// SIMATIC S7-200 project (STEP 7-Micro/WIN), CPU 226 CN REL 02.01

SYMBOL_TABLE USER1
Sens_Origen      I0.0     // Sensor inductivo origen servo (usado por libreria MAP_SERV para homing)
FC_Derecha       I0.1     // Final de carrera derecha (Fwd_Limit para Q0_0_CTRL)
FC_Izquierda     I0.2     // Final de carrera izquierda (Rev_Limit para Q0_0_CTRL)
CilV_Abajo       I0.3     // Sensor brazo retraido (abajo)
CilV_Arriba      I0.4     // Sensor brazo extendido (arriba)
Giro_Izquierda   I0.5     // Sensor rotatorio posicion izquierda (antihorario)
Giro_Derecha     I0.6     // Sensor rotatorio posicion derecha (horario)
CilDV_Ext        I0.7     // Sensor doble vastago extendido
CilDV_Ret        I1.0     // Sensor doble vastago retraido
Pinza_Cer        I1.1     // Sensor pinza cerrada
Estado_Servo     I1.2     // Estado driver servo (1=Ready 0=Alarma)
Btn_Paro         I2.4     // Pulsador rojo de paro
Btn_Marcha       I2.5     // Pulsador amarillo de marcha
Seta_Emerg       I2.6     // Seta de emergencia (NC - 0=emergencia activa)
Selector         I2.7     // Selector rotatorio de modo
Servo_Pulsos     Q0.0     // Salida PTO tren de pulsos al driver servo
Servo_Dir        Q0.2     // Salida direccion al driver servo
V_Cil_Vert       Q0.3     // Valvula elevar brazo neumatico (activo=arriba inactivo=baja)
V_Giro_AH        Q0.4     // Valvula rotatorio antihorario (destino Seleccion)
V_Giro_H         Q0.5     // Valvula rotatorio horario (destino Procesamiento y Ensamblaje)
V_Cil_DV         Q0.6     // Valvula doble vastago (extender)
V_Pinza_Abre     Q0.7     // Valvula pinza abre
V_Pinza_Cierra   Q1.0     // Valvula pinza cierra
Lamp_Amarilla    Q1.5     // Lampara amarilla - parada pendiente o homing activo
Lamp_Verde       Q1.6     // Lampara verde - ciclo de tarea en ejecucion
Lamp_Roja        Q1.7     // Lampara roja - reposo esperando solicitud
P_Hom_Espera     M5.0     // Plaza Homing_Espera - estado inicial al arranque o tras emergencia
P_Hom_Activo     M5.1     // Plaza Homing_Activo - servo buscando origen
P0_Brazo_Libre   M0.0     // Plaza P0 - Reposo. Brazo disponible para nueva tarea
P1_Req_A_P       M0.1     // Plaza P1 - Solicitud activa Alimentacion -> Procesamiento (inyectable Modbus)
P2_Req_P_E       M0.2     // Plaza P2 - Solicitud activa Procesamiento -> Ensamblaje (inyectable Modbus)
P3_Req_E_S       M0.3     // Plaza P3 - Solicitud activa Ensamblaje -> Seleccion (inyectable Modbus)
P10_Viaje_Ori    M1.0     // Plaza P10 - Servo viajando a coordenada de recogida
P11a_Rot_Ori     M1.1     // Plaza P11a - Orientando garra en posicion de recogida
P11b_DV_Ext      M1.2     // Plaza P11b - Extendiendo doble vastago en pick
P11c_Cil_Baj     M1.3     // Plaza P11c - Bajando brazo en pick
P11d_Pinza_Cer   M1.4     // Plaza P11d - Cerrando pinza (agarrando pieza)
P11e_Cil_Arr     M1.5     // Plaza P11e - Subiendo brazo con pieza
P11f_DV_Ret      M1.6     // Plaza P11f - Retrayendo doble vastago (pick completo)
P12_Viaje_Des    M1.7     // Plaza P12 - Servo viajando a coordenada de entrega
P13a_Rot_Des     M2.0     // Plaza P13a - Orientando garra en posicion de entrega
P13b_DV_Ext      M2.1     // Plaza P13b - Extendiendo doble vastago en place
P13c_Cil_Baj     M2.2     // Plaza P13c - Bajando brazo en place
P13d_Pinza_Ab    M8.0     // Plaza P13d - Abriendo pinza (liberando pieza)
P13e_Cil_Arr     M8.1     // Plaza P13e - Subiendo brazo tras soltar
P13f_DV_Ret      M3.5     // Plaza P13f - Retrayendo doble vastago (place completo)
P14_Finalizar    M3.6     // Plaza P14 - Liberando brazo y limpiando solicitud
Ev_Marcha_Flanco M6.0     // Evento - Flanco subida boton marcha (autorreset en P0)
Ev_Paro_Flanco   M6.1     // Evento - Flanco subida boton paro (bloquea inicio nuevo ciclo)
Ev_CilV_Abajo    M2.3     // Evento - Sensor brazo abajo
Ev_CilV_Arriba   M2.4     // Evento - Sensor brazo arriba
Ev_Giro_Izq      M2.5     // Evento - Sensor rotatorio posicion izquierda
Ev_Giro_Der      M2.6     // Evento - Sensor rotatorio posicion derecha (horario)
Ev_CilDV_Ext     M2.7     // Evento - Sensor doble vastago extendido
Ev_CilDV_Ret     M3.0     // Evento - Sensor doble vastago retraido
Ev_Pinza_Cer     M3.1     // Evento - Pinza cerrada
Ev_Move_Done     M3.2     // Evento - Flag Done libreria MAP_SERV (posicion alcanzada)
Ev_Origen_Det    M3.3     // Evento - Sensor I0.0 origen detectado (usado en homing)
Ev_Servo_OK      M3.4     // Evento - Driver servo listo (I1.2=1)
T_Homing_Start   M4.0     // Disparo - Iniciar secuencia de homing
T_Homing_Done    M4.1     // Disparo - Homing completado sensor origen detectado
T_Acept_ES       M4.2     // Disparo - Aceptar tarea E->S (Prioridad 1 alta)
T_Acept_PE       M4.3     // Disparo - Aceptar tarea P->E (Prioridad 2 media)
T_Acept_AP       M4.4     // Disparo - Aceptar tarea A->P (Prioridad 3 baja)
T_Origen_OK      M4.5     // Disparo - Servo llego a coordenada de recogida
T_Rot_Ori_OK     M4.6     // Disparo - Garra orientada en posicion de recogida
T_DV_Ext_Pick    M4.7     // Disparo - Doble vastago extendido en pick
T_CilV_Baj_Pick  M5.2     // Disparo - Brazo abajo en pick
T_Pinza_Cer      M5.3     // Disparo - Pinza cerrada agarre confirmado
T_CilV_Arr_Pick  M5.4     // Disparo - Brazo arriba con pieza en pick
T_DV_Ret_Pick    M5.5     // Disparo - Doble vastago retraido pick completo
T_Destino_OK     M5.6     // Disparo - Servo llego a coordenada de entrega
T_Rot_Des_OK     M5.7     // Disparo - Garra orientada en posicion de entrega
T_DV_Ext_Place   M6.2     // Disparo - Doble vastago extendido en place
T_CilV_Baj_Place M6.3     // Disparo - Brazo abajo en place
T_Pinza_Ab       M6.4     // Disparo - Pinza abierta pieza liberada
T_CilV_Arr_Place M6.5     // Disparo - Brazo arriba tras soltar en place
T_DV_Ret_Place   M6.6     // Disparo - Doble vastago retraido place completo
T_Tarea_Fin      M6.7     // Disparo - Liberar brazo y volver a reposo
Ctx_Tarea_AP     M7.0     // Contexto tarea activa - Alimentacion -> Procesamiento
Ctx_Tarea_PE     M7.1     // Contexto tarea activa - Procesamiento -> Ensamblaje
Ctx_Tarea_ES     M7.2     // Contexto tarea activa - Ensamblaje -> Seleccion
Home_Done        V221.0   // Bit Done libreria MAP_SERV (busqueda de origen alcanzada)
Home_error       V221.1   // Bit Error libreria MAP_SERV (avisa si hubo un error en la busqueda de origen)
Servo_Exec       V220.0   // Bit interno - Comando ejecutar movimiento (nivel)
Servo_Done       V220.1   // Bit Done libreria MAP_SERV (posicion alcanzada)
Servo_Err        V220.2   // Bit Error libreria MAP_SERV
Servo_Execute_Pulse V220.4   // Bit pulso EXECUTE un scan para MoveAbsolute
Servo_C_Pos      VD34     // Posicion actual del servo en pulsos (salida Q0_0_CTRL)
Coord_Target     VD200    // Coordenada destino activa cargada antes de MoveAbsolute
Coord_Alim       VD204    // Coordenada estacion Alimentacion (pulsos)
Coord_Proc       VD208    // Coordenada estacion Procesamiento (pulsos)
Coord_Ensa       VD212    // Coordenada estacion Ensamblaje (pulsos)
Coord_Sele       VD216    // Coordenada estacion Seleccion (pulsos)
net_cycle        M10.0    // network cycle (PPI)
net_error        M10.1    // network error (PPI)
done_modbus      M10.2    // marca done para libreria modbus (init)
error_modbus     VB26     // byte de error para libreria modbus (init)
done_modbus2     M10.3    // marca done para libreria modbus
error_modbus2    VB30     // byte de error para libreria modbus
Pos_Alim         VD10     // Posicion Alimentacion (buffer para la carga dinamica de la posicion)
Pos_Proc         VD14     // Posicion Procesamiento (buffer para la carga dinamica de la posicion)
Pos_Ensa         VD18     // Posicion Ensamblaje (buffer para la carga dinamica de la posicion)
Pos_Sele         VD22     // Posicion Seleccion (buffer para la carga dinamica de la posicion)
Sol_AP           V0.0     // Solicitud Alimentacion a Procesamiento
Ack_AP           V1.0     // Reconocimiento AP
Sol_PE           V2.0     // Solicitud Procesamiento a Ensamblaje
Ack_PE           V3.0     // Reconocimiento PE
Sol_ES           V4.0     // Solicitud Ensamblaje a Seleccion
Ack_ES           V5.0     // Reconocimiento ES
Ack_MA           V0.1     // Reconocimiento marcha Unidad de Alimentacion
Marcha_A         V1.1     // Solicitud de marcha para la Unidad de Alimentacion
Ack_MP           V2.1     // Reconocimiento marcha Unidad de Procesammiento
Marcha_P         V3.1     // Solicitud de marcha para la Unidad de Procesamiento
Ack_ME           V4.1     // Reconocimiento marcha Unidad de Ensamblaje
Marcha_E         V5.1     // Solicitud de marcha para la Unidad de Ensamblaje
Ack_MS           V6.1     // Reconocimiento marcha Unidad de Seleccion
Marcha_S         V7.1     // Solicitud de marcha para la Unidad de Seleccion
Alim_OK          V0.2     // Unidad de Alimentacion disponible
Proc_OK          V2.2     // Unidad de Procesamiento disponible
Ens_OK           V4.2     // Unidad de Ensamblaje disponible
Sel_OK           V6.2     // Unidad de Seleccion disponible
Pieza_Metal      V6.3     // Pieza identificada por la unidad de seleccion es totalmente metalica
Pieza_Mixta      V6.4     // Pieza identificada por la unidad de seleccion es totalmente mixta
Pieza_Plastica   V6.5     // Pieza identificada por la unidad de seleccion es totalmente plastica
END_SYMBOL_TABLE

SYMBOL_TABLE S7-200 Symbols
Always_On        SM0.0    // 始终接通为 ON
First_Scan_On    SM0.1    // 仅第一个扫描周期中接通为 ON
END_SYMBOL_TABLE

ORGANIZATION_BLOCK MAIN:OB1
TITLE=UNIDAD DE TRANSPORTE - RED DE PETRI CIPN
//  ===========================================================
//  MODULO 0: SEGURIDAD - Evaluado primero en cada scan.
//  Si Seta = 0 (NC abierta): reset total, fuerza P_Homing,
//  apaga salidas neumaticas. El servo se detiene porque
//  Q0_0_CTRL deja de recibir EXECUTE.
//  ===========================================================
BEGIN
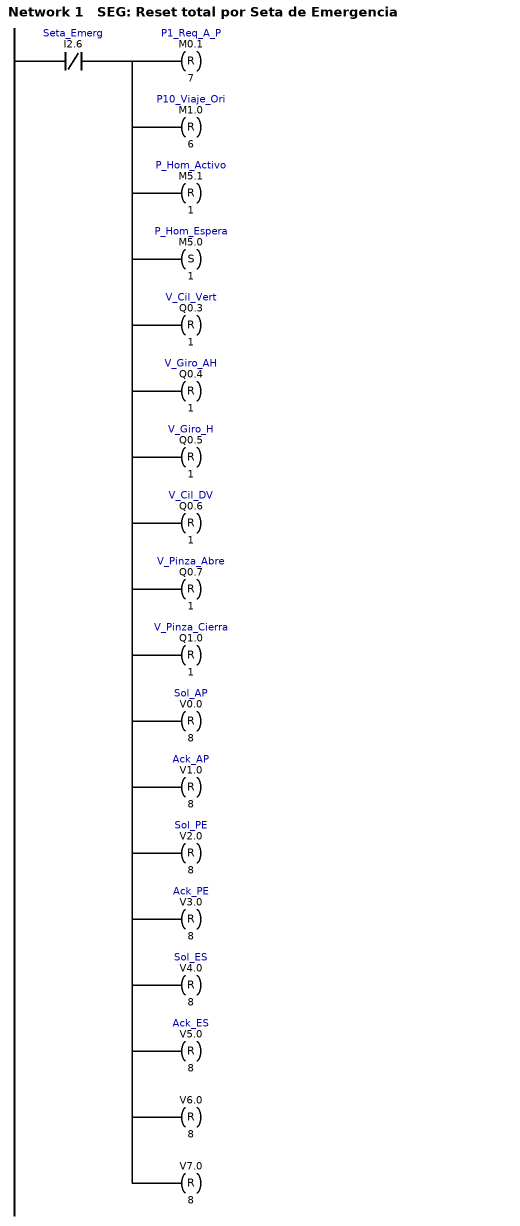
Network 1 //  SEG: Reset total por Seta de Emergencia
LDN    Seta_Emerg:I2.6
R      P1_Req_A_P:M0.1, 7
R      P10_Viaje_Ori:M1.0, 6
R      P_Hom_Activo:M5.1, 1
S      P_Hom_Espera:M5.0, 1
R      V_Cil_Vert:Q0.3, 1
R      V_Giro_AH:Q0.4, 1
R      V_Giro_H:Q0.5, 1
R      V_Cil_DV:Q0.6, 1
R      V_Pinza_Abre:Q0.7, 1
R      V_Pinza_Cierra:Q1.0, 1
R      Sol_AP:V0.0, 8
R      Ack_AP:V1.0, 8
R      Sol_PE:V2.0, 8
R      Ack_PE:V3.0, 8
R      Sol_ES:V4.0, 8
R      Ack_ES:V5.0, 8
R      V6.0, 8
R      V7.0, 8
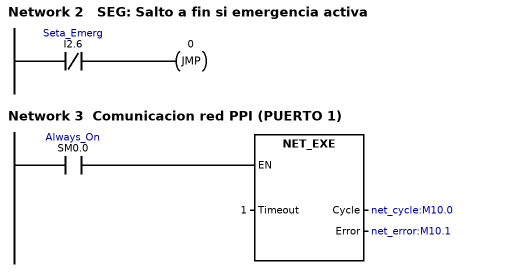
Network 2 //  SEG: Salto a fin si emergencia activa
LDN    Seta_Emerg:I2.6
JMP    0
Network 3 // Comunicacion red PPI (PUERTO 1)
LD     Always_On:SM0.0
CALL   NET_EXE:SBR6, 1, net_cycle:M10.0, net_error:M10.1
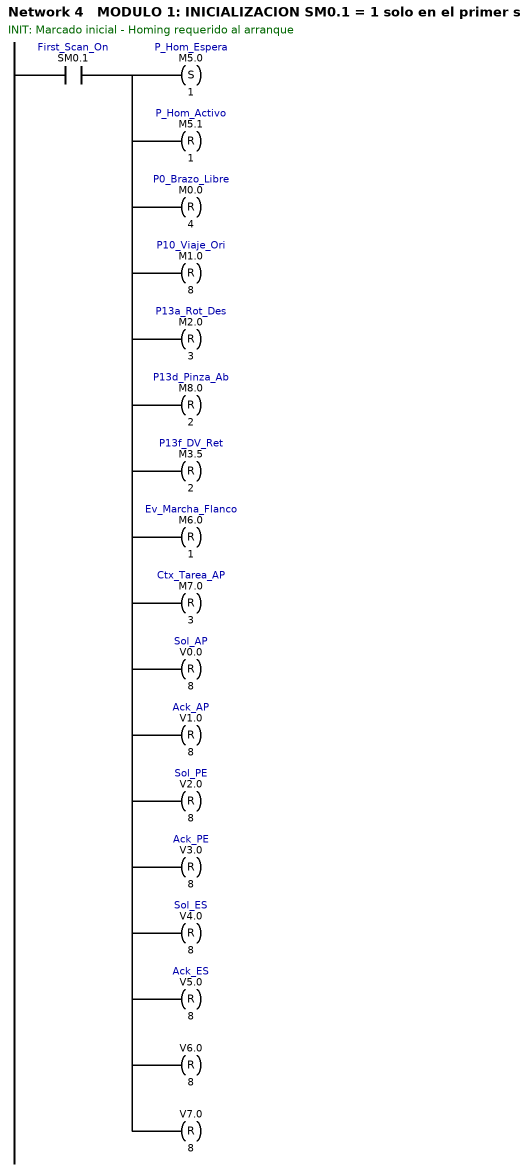
Network 4 //  MODULO 1: INICIALIZACION
SM0.1 = 1 solo en el primer scan.
Marcado inicial: P_Homing activo (M5.0).
El brazo debe calibrarse antes de aceptar cualquier tarea.
Coordenadas de estaciones cargadas en VD fijos.
// INIT: Marcado inicial - Homing requerido al arranque
LD     First_Scan_On:SM0.1
S      P_Hom_Espera:M5.0, 1
R      P_Hom_Activo:M5.1, 1
R      P0_Brazo_Libre:M0.0, 4
R      P10_Viaje_Ori:M1.0, 8
R      P13a_Rot_Des:M2.0, 3
R      P13d_Pinza_Ab:M8.0, 2
R      P13f_DV_Ret:M3.5, 2
R      Ev_Marcha_Flanco:M6.0, 1
R      Ctx_Tarea_AP:M7.0, 3
R      Sol_AP:V0.0, 8
R      Ack_AP:V1.0, 8
R      Sol_PE:V2.0, 8
R      Ack_PE:V3.0, 8
R      Sol_ES:V4.0, 8
R      Ack_ES:V5.0, 8
R      V6.0, 8
R      V7.0, 8
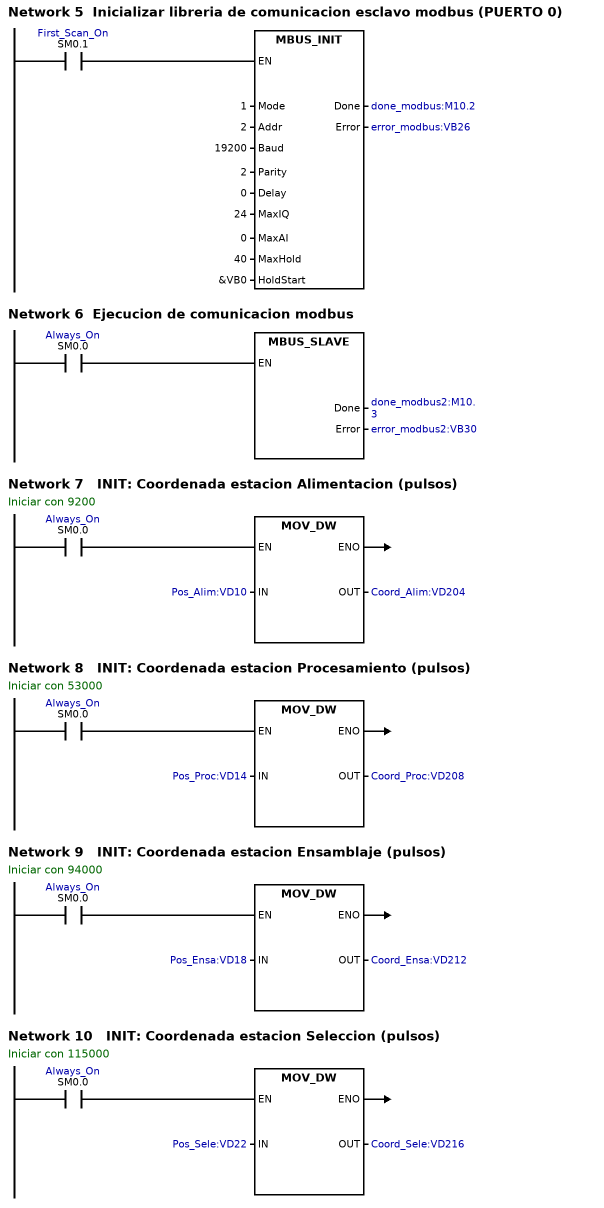
Network 5 // Inicializar libreria de comunicacion esclavo modbus (PUERTO 0)
LD     First_Scan_On:SM0.1
CALL   MBUS_INIT:SBR7, 1, 2, 19200, 2, 0, 24, 0, 40, &VB0, done_modbus:M10.2, error_modbus:VB26
Network 6 // Ejecucion de comunicacion modbus
LD     Always_On:SM0.0
CALL   MBUS_SLAVE:SBR8, done_modbus2:M10.3, error_modbus2:VB30
Network 7 //  INIT: Coordenada estacion Alimentacion (pulsos)
// Iniciar con 9200
LD     Always_On:SM0.0
MOVD   Pos_Alim:VD10, Coord_Alim:VD204
Network 8 //  INIT: Coordenada estacion Procesamiento (pulsos)
// Iniciar con 53000
LD     Always_On:SM0.0
MOVD   Pos_Proc:VD14, Coord_Proc:VD208
Network 9 //  INIT: Coordenada estacion Ensamblaje (pulsos)
// Iniciar con 94000
LD     Always_On:SM0.0
MOVD   Pos_Ensa:VD18, Coord_Ensa:VD212
Network 10 //  INIT: Coordenada estacion Seleccion (pulsos)
// Iniciar con 115000
LD     Always_On:SM0.0
MOVD   Pos_Sele:VD22, Coord_Sele:VD216
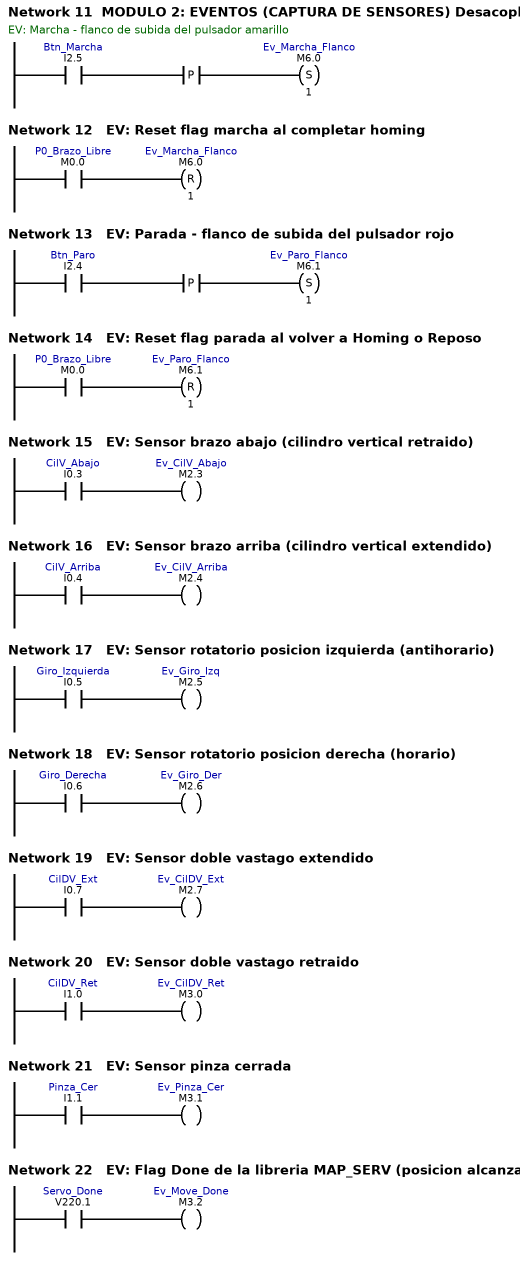
Network 11 // MODULO 2: EVENTOS (CAPTURA DE SENSORES)
Desacopla la logica secuencial de las senales fisicas.
M5.x reservado para estados de Homing y sistema.
M2.x / M3.x para eventos de sensores.
// EV: Marcha - flanco de subida del pulsador amarillo
LD     Btn_Marcha:I2.5
EU
S      Ev_Marcha_Flanco:M6.0, 1
Network 12 //  EV: Reset flag marcha al completar homing
LD     P0_Brazo_Libre:M0.0
R      Ev_Marcha_Flanco:M6.0, 1
Network 13 //  EV: Parada - flanco de subida del pulsador rojo
LD     Btn_Paro:I2.4
EU
S      Ev_Paro_Flanco:M6.1, 1
Network 14 //  EV: Reset flag parada al volver a Homing o Reposo
LD     P0_Brazo_Libre:M0.0
R      Ev_Paro_Flanco:M6.1, 1
Network 15 //  EV: Sensor brazo abajo (cilindro vertical retraido)
LD     CilV_Abajo:I0.3
=      Ev_CilV_Abajo:M2.3
Network 16 //  EV: Sensor brazo arriba (cilindro vertical extendido)
LD     CilV_Arriba:I0.4
=      Ev_CilV_Arriba:M2.4
Network 17 //  EV: Sensor rotatorio posicion izquierda (antihorario)
LD     Giro_Izquierda:I0.5
=      Ev_Giro_Izq:M2.5
Network 18 //  EV: Sensor rotatorio posicion derecha (horario)
LD     Giro_Derecha:I0.6
=      Ev_Giro_Der:M2.6
Network 19 //  EV: Sensor doble vastago extendido
LD     CilDV_Ext:I0.7
=      Ev_CilDV_Ext:M2.7
Network 20 //  EV: Sensor doble vastago retraido
LD     CilDV_Ret:I1.0
=      Ev_CilDV_Ret:M3.0
Network 21 //  EV: Sensor pinza cerrada
LD     Pinza_Cer:I1.1
=      Ev_Pinza_Cer:M3.1
Network 22 //  EV: Flag Done de la libreria MAP_SERV (posicion alcanzada)
LD     Servo_Done:V220.1
=      Ev_Move_Done:M3.2
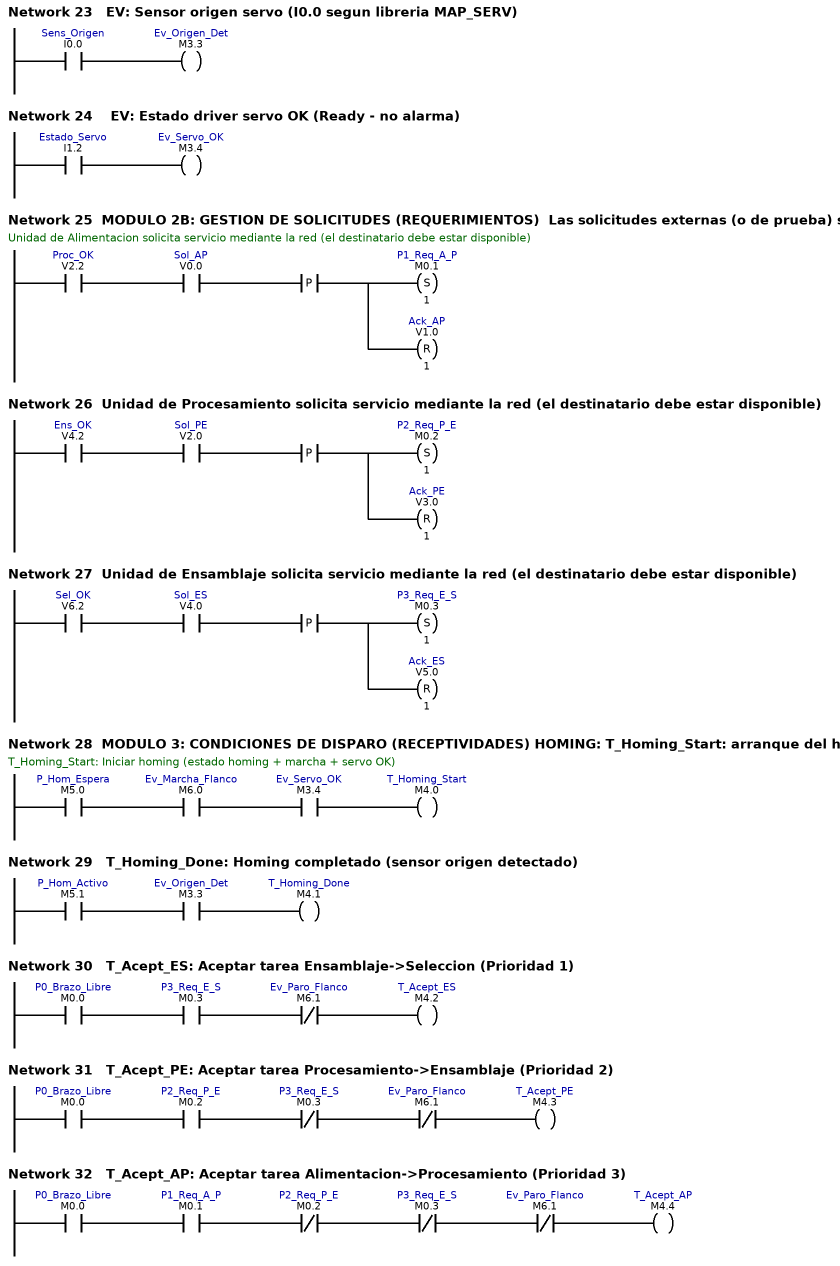
Network 23 //  EV: Sensor origen servo (I0.0 segun libreria MAP_SERV)
LD     Sens_Origen:I0.0
=      Ev_Origen_Det:M3.3
Network 24 //   EV: Estado driver servo OK (Ready - no alarma)
LD     Estado_Servo:I1.2
=      Ev_Servo_OK:M3.4
Network 25 // MODULO 2B: GESTION DE SOLICITUDES (REQUERIMIENTOS)
 Las solicitudes externas (o de prueba) se inyectan en
 M0.1, M0.2, M0.3 desde fuera (Modbus, HMI, o prueba manual).
 Este bloque las protege: solo se aceptan si el sistema
 esta en Reposo (P0 = M0.0 activo)
// Unidad de Alimentacion solicita servicio mediante la red (el destinatario debe estar disponible)
LD     Proc_OK:V2.2
A      Sol_AP:V0.0
EU
S      P1_Req_A_P:M0.1, 1
R      Ack_AP:V1.0, 1
Network 26 // Unidad de Procesamiento solicita servicio mediante la red (el destinatario debe estar disponible)
LD     Ens_OK:V4.2
A      Sol_PE:V2.0
EU
S      P2_Req_P_E:M0.2, 1
R      Ack_PE:V3.0, 1
Network 27 // Unidad de Ensamblaje solicita servicio mediante la red (el destinatario debe estar disponible)
LD     Sel_OK:V6.2
A      Sol_ES:V4.0
EU
S      P3_Req_E_S:M0.3, 1
R      Ack_ES:V5.0, 1
Network 28 // MODULO 3: CONDICIONES DE DISPARO (RECEPTIVIDADES)
HOMING:
T_Homing_Start: arranque del homing (marcha presionada)
T_Homing_Done:  sensor origen detectado
ACEPTACION DE TAREA (priorizadas, mutuamente excluyentes):
T_Acept_ES: P0 AND P3           (Prioridad 1 - Alta)
T_Acept_PE: P0 AND P2 AND !P3   (Prioridad 2 - Media)
T_Acept_AP: P0 AND P1 AND !P2 !P3 (Prioridad 3 - Baja)
CICLO DE TAREA:
Sub-plazas Pick (P11a..P11e) y Place (P13a..P13e)
para modelar los 5 pasos de cada secuencia.
//  T_Homing_Start: Iniciar homing (estado homing + marcha + servo OK)
LD     P_Hom_Espera:M5.0
A      Ev_Marcha_Flanco:M6.0
A      Ev_Servo_OK:M3.4
=      T_Homing_Start:M4.0
Network 29 //  T_Homing_Done: Homing completado (sensor origen detectado)
LD     P_Hom_Activo:M5.1
A      Ev_Origen_Det:M3.3
=      T_Homing_Done:M4.1
Network 30 //  T_Acept_ES: Aceptar tarea Ensamblaje->Seleccion (Prioridad 1)
LD     P0_Brazo_Libre:M0.0
A      P3_Req_E_S:M0.3
AN     Ev_Paro_Flanco:M6.1
=      T_Acept_ES:M4.2
Network 31 //  T_Acept_PE: Aceptar tarea Procesamiento->Ensamblaje (Prioridad 2)
LD     P0_Brazo_Libre:M0.0
A      P2_Req_P_E:M0.2
AN     P3_Req_E_S:M0.3
AN     Ev_Paro_Flanco:M6.1
=      T_Acept_PE:M4.3
Network 32 //  T_Acept_AP: Aceptar tarea Alimentacion->Procesamiento (Prioridad 3)
LD     P0_Brazo_Libre:M0.0
A      P1_Req_A_P:M0.1
AN     P2_Req_P_E:M0.2
AN     P3_Req_E_S:M0.3
AN     Ev_Paro_Flanco:M6.1
=      T_Acept_AP:M4.4
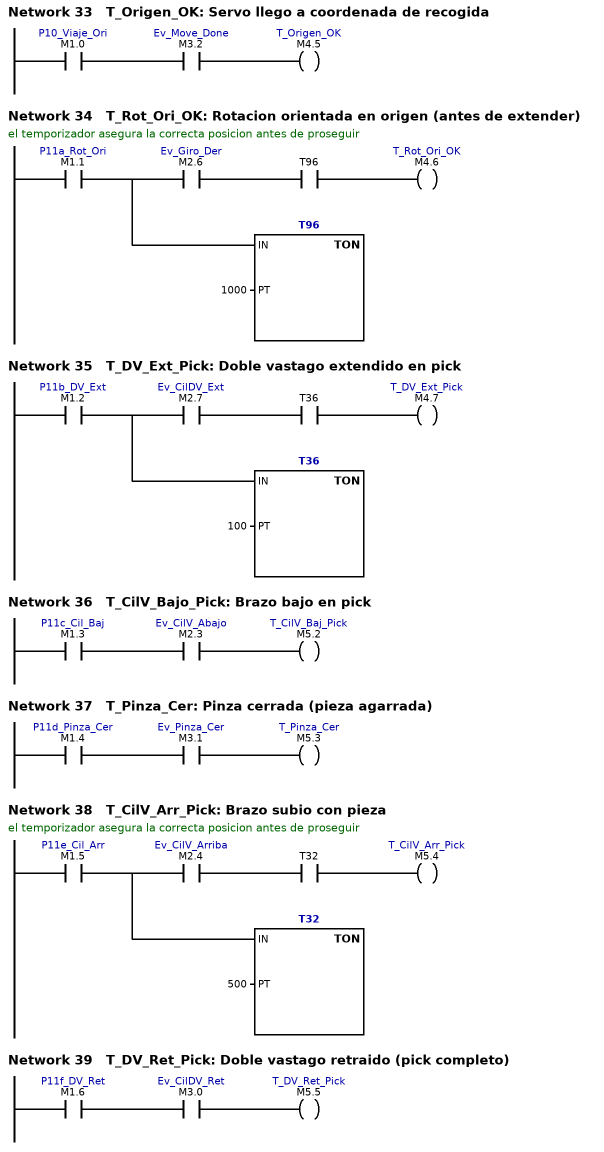
Network 33 //  T_Origen_OK: Servo llego a coordenada de recogida
LD     P10_Viaje_Ori:M1.0
A      Ev_Move_Done:M3.2
=      T_Origen_OK:M4.5
Network 34 //  T_Rot_Ori_OK: Rotacion orientada en origen (antes de extender)
// el temporizador asegura la correcta posicion antes de proseguir
LD     P11a_Rot_Ori:M1.1
LPS
A      Ev_Giro_Der:M2.6
A      T96
=      T_Rot_Ori_OK:M4.6
LPP
TON    T96, 1000
Network 35 //  T_DV_Ext_Pick: Doble vastago extendido en pick
LD     P11b_DV_Ext:M1.2
LPS
A      Ev_CilDV_Ext:M2.7
A      T36
=      T_DV_Ext_Pick:M4.7
LPP
TON    T36, 100
Network 36 //  T_CilV_Bajo_Pick: Brazo bajo en pick
LD     P11c_Cil_Baj:M1.3
A      Ev_CilV_Abajo:M2.3
=      T_CilV_Baj_Pick:M5.2
Network 37 //  T_Pinza_Cer: Pinza cerrada (pieza agarrada)
LD     P11d_Pinza_Cer:M1.4
A      Ev_Pinza_Cer:M3.1
=      T_Pinza_Cer:M5.3
Network 38 //  T_CilV_Arr_Pick: Brazo subio con pieza
// el temporizador asegura la correcta posicion antes de proseguir
LD     P11e_Cil_Arr:M1.5
LPS
A      Ev_CilV_Arriba:M2.4
A      T32
=      T_CilV_Arr_Pick:M5.4
LPP
TON    T32, 500
Network 39 //  T_DV_Ret_Pick: Doble vastago retraido (pick completo)
LD     P11f_DV_Ret:M1.6
A      Ev_CilDV_Ret:M3.0
=      T_DV_Ret_Pick:M5.5
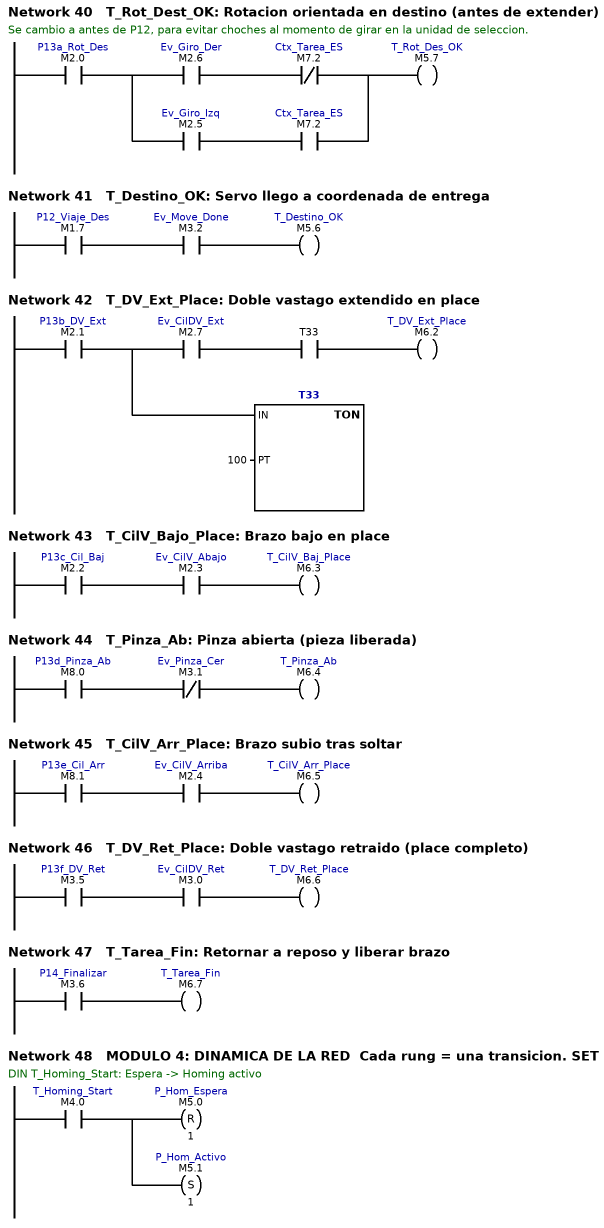
Network 40 //  T_Rot_Dest_OK: Rotacion orientada en destino (antes de extender)
// Se cambio a antes de P12, para evitar choches al momento de girar en la unidad de seleccion.
LD     P13a_Rot_Des:M2.0
LD     Ev_Giro_Der:M2.6
AN     Ctx_Tarea_ES:M7.2
LD     Ev_Giro_Izq:M2.5
A      Ctx_Tarea_ES:M7.2
OLD
ALD
=      T_Rot_Des_OK:M5.7
Network 41 //  T_Destino_OK: Servo llego a coordenada de entrega
LD     P12_Viaje_Des:M1.7
A      Ev_Move_Done:M3.2
=      T_Destino_OK:M5.6
Network 42 //  T_DV_Ext_Place: Doble vastago extendido en place
LD     P13b_DV_Ext:M2.1
LPS
A      Ev_CilDV_Ext:M2.7
A      T33
=      T_DV_Ext_Place:M6.2
LPP
TON    T33, 100
Network 43 //  T_CilV_Bajo_Place: Brazo bajo en place
LD     P13c_Cil_Baj:M2.2
A      Ev_CilV_Abajo:M2.3
=      T_CilV_Baj_Place:M6.3
Network 44 //  T_Pinza_Ab: Pinza abierta (pieza liberada)
LD     P13d_Pinza_Ab:M8.0
AN     Ev_Pinza_Cer:M3.1
=      T_Pinza_Ab:M6.4
Network 45 //  T_CilV_Arr_Place: Brazo subio tras soltar
LD     P13e_Cil_Arr:M8.1
A      Ev_CilV_Arriba:M2.4
=      T_CilV_Arr_Place:M6.5
Network 46 //  T_DV_Ret_Place: Doble vastago retraido (place completo)
LD     P13f_DV_Ret:M3.5
A      Ev_CilDV_Ret:M3.0
=      T_DV_Ret_Place:M6.6
Network 47 //  T_Tarea_Fin: Retornar a reposo y liberar brazo
//  
LD     P14_Finalizar:M3.6
=      T_Tarea_Fin:M6.7
Network 48 //  MODULO 4: DINAMICA DE LA RED
 Cada rung = una transicion. SET destino, RESET origen.
 El marcado de contexto (cual solicitud se esta atendiendo)
 se guarda en M7.0 (es A->P), M7.1 (es P->E), M7.2 (es E->S).
 La orientacion de garra se decide por M7.2 (Seleccion=AH).
// DIN T_Homing_Start: Espera -> Homing activo
LD     T_Homing_Start:M4.0
R      P_Hom_Espera:M5.0, 1
S      P_Hom_Activo:M5.1, 1
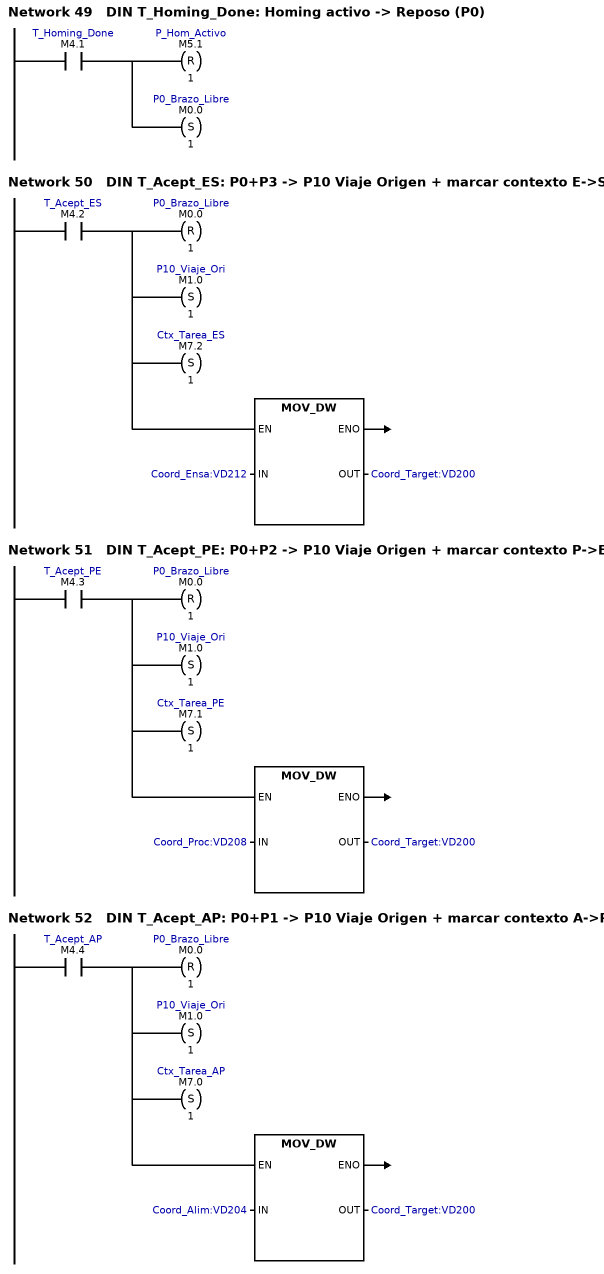
Network 49 //  DIN T_Homing_Done: Homing activo -> Reposo (P0)
LD     T_Homing_Done:M4.1
R      P_Hom_Activo:M5.1, 1
S      P0_Brazo_Libre:M0.0, 1
Network 50 //  DIN T_Acept_ES: P0+P3 -> P10 Viaje Origen + marcar contexto E->S
LD     T_Acept_ES:M4.2
R      P0_Brazo_Libre:M0.0, 1
S      P10_Viaje_Ori:M1.0, 1
S      Ctx_Tarea_ES:M7.2, 1
MOVD   Coord_Ensa:VD212, Coord_Target:VD200
Network 51 //  DIN T_Acept_PE: P0+P2 -> P10 Viaje Origen + marcar contexto P->E
LD     T_Acept_PE:M4.3
R      P0_Brazo_Libre:M0.0, 1
S      P10_Viaje_Ori:M1.0, 1
S      Ctx_Tarea_PE:M7.1, 1
MOVD   Coord_Proc:VD208, Coord_Target:VD200
Network 52 //  DIN T_Acept_AP: P0+P1 -> P10 Viaje Origen + marcar contexto A->P
LD     T_Acept_AP:M4.4
R      P0_Brazo_Libre:M0.0, 1
S      P10_Viaje_Ori:M1.0, 1
S      Ctx_Tarea_AP:M7.0, 1
MOVD   Coord_Alim:VD204, Coord_Target:VD200
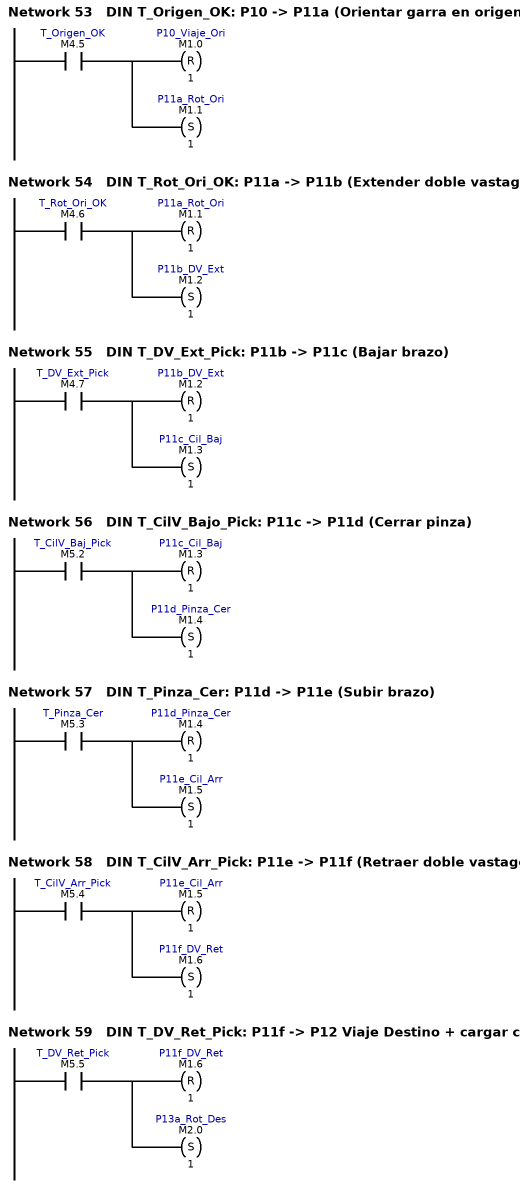
Network 53 //  DIN T_Origen_OK: P10 -> P11a (Orientar garra en origen)
LD     T_Origen_OK:M4.5
R      P10_Viaje_Ori:M1.0, 1
S      P11a_Rot_Ori:M1.1, 1
Network 54 //  DIN T_Rot_Ori_OK: P11a -> P11b (Extender doble vastago)
LD     T_Rot_Ori_OK:M4.6
R      P11a_Rot_Ori:M1.1, 1
S      P11b_DV_Ext:M1.2, 1
Network 55 //  DIN T_DV_Ext_Pick: P11b -> P11c (Bajar brazo)
LD     T_DV_Ext_Pick:M4.7
R      P11b_DV_Ext:M1.2, 1
S      P11c_Cil_Baj:M1.3, 1
Network 56 //  DIN T_CilV_Bajo_Pick: P11c -> P11d (Cerrar pinza)
LD     T_CilV_Baj_Pick:M5.2
R      P11c_Cil_Baj:M1.3, 1
S      P11d_Pinza_Cer:M1.4, 1
Network 57 //  DIN T_Pinza_Cer: P11d -> P11e (Subir brazo)
LD     T_Pinza_Cer:M5.3
R      P11d_Pinza_Cer:M1.4, 1
S      P11e_Cil_Arr:M1.5, 1
Network 58 //  DIN T_CilV_Arr_Pick: P11e -> P11f (Retraer doble vastago)
LD     T_CilV_Arr_Pick:M5.4
R      P11e_Cil_Arr:M1.5, 1
S      P11f_DV_Ret:M1.6, 1
Network 59 //  DIN T_DV_Ret_Pick: P11f -> P12 Viaje Destino + cargar coord destino
LD     T_DV_Ret_Pick:M5.5
R      P11f_DV_Ret:M1.6, 1
S      P13a_Rot_Des:M2.0, 1
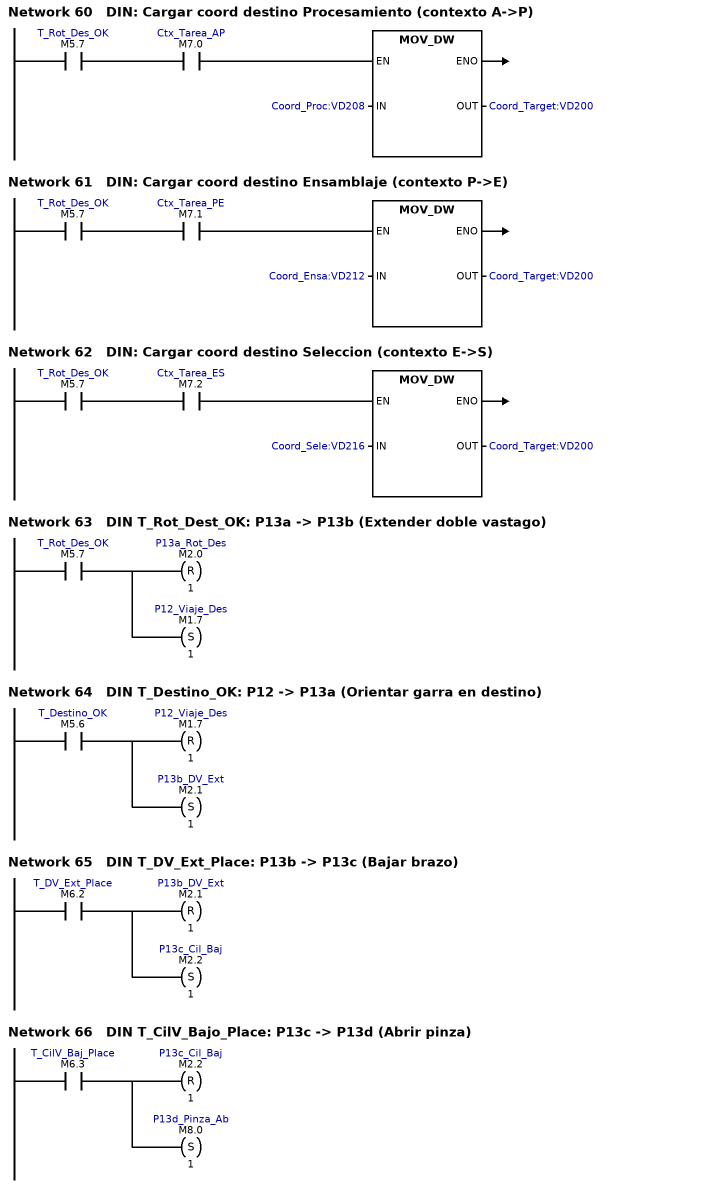
Network 60 //  DIN: Cargar coord destino Procesamiento (contexto A->P)
LD     T_Rot_Des_OK:M5.7
A      Ctx_Tarea_AP:M7.0
MOVD   Coord_Proc:VD208, Coord_Target:VD200
Network 61 //  DIN: Cargar coord destino Ensamblaje (contexto P->E)
LD     T_Rot_Des_OK:M5.7
A      Ctx_Tarea_PE:M7.1
MOVD   Coord_Ensa:VD212, Coord_Target:VD200
Network 62 //  DIN: Cargar coord destino Seleccion (contexto E->S)
LD     T_Rot_Des_OK:M5.7
A      Ctx_Tarea_ES:M7.2
MOVD   Coord_Sele:VD216, Coord_Target:VD200
Network 63 //  DIN T_Rot_Dest_OK: P13a -> P13b (Extender doble vastago)
LD     T_Rot_Des_OK:M5.7
R      P13a_Rot_Des:M2.0, 1
S      P12_Viaje_Des:M1.7, 1
Network 64 //  DIN T_Destino_OK: P12 -> P13a (Orientar garra en destino)
LD     T_Destino_OK:M5.6
R      P12_Viaje_Des:M1.7, 1
S      P13b_DV_Ext:M2.1, 1
Network 65 //  DIN T_DV_Ext_Place: P13b -> P13c (Bajar brazo)
LD     T_DV_Ext_Place:M6.2
R      P13b_DV_Ext:M2.1, 1
S      P13c_Cil_Baj:M2.2, 1
Network 66 //  DIN T_CilV_Bajo_Place: P13c -> P13d (Abrir pinza)
LD     T_CilV_Baj_Place:M6.3
R      P13c_Cil_Baj:M2.2, 1
S      P13d_Pinza_Ab:M8.0, 1
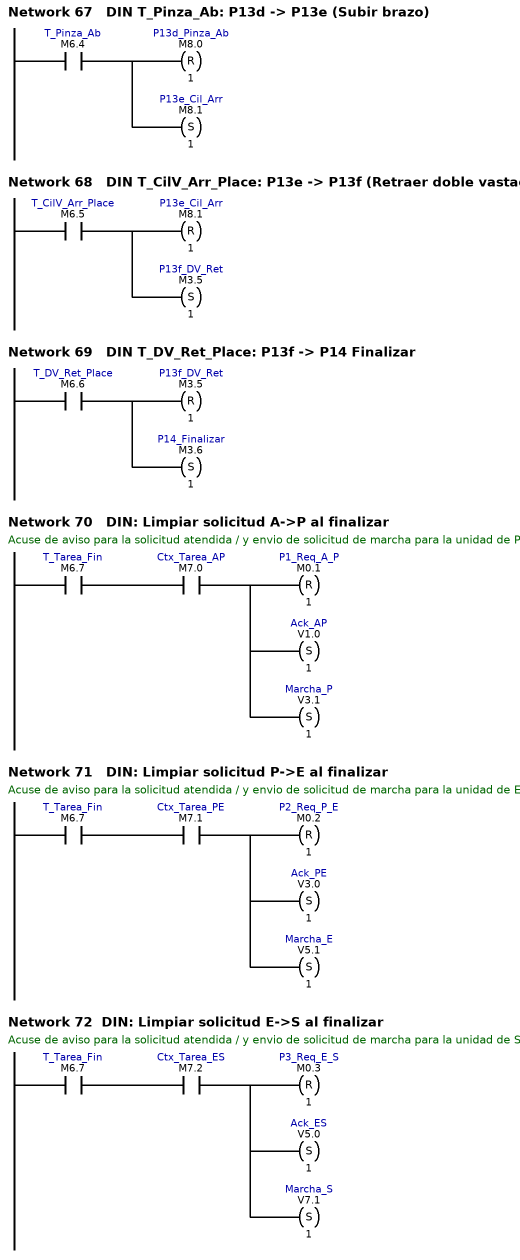
Network 67 //  DIN T_Pinza_Ab: P13d -> P13e (Subir brazo)
LD     T_Pinza_Ab:M6.4
R      P13d_Pinza_Ab:M8.0, 1
S      P13e_Cil_Arr:M8.1, 1
Network 68 //  DIN T_CilV_Arr_Place: P13e -> P13f (Retraer doble vastago)
LD     T_CilV_Arr_Place:M6.5
R      P13e_Cil_Arr:M8.1, 1
S      P13f_DV_Ret:M3.5, 1
Network 69 //  DIN T_DV_Ret_Place: P13f -> P14 Finalizar
LD     T_DV_Ret_Place:M6.6
R      P13f_DV_Ret:M3.5, 1
S      P14_Finalizar:M3.6, 1
Network 70 //  DIN: Limpiar solicitud A->P al finalizar
// Acuse de aviso para la solicitud atendida
// y envio de solicitud de marcha para la unidad de Procesamiento
LD     T_Tarea_Fin:M6.7
A      Ctx_Tarea_AP:M7.0
R      P1_Req_A_P:M0.1, 1
S      Ack_AP:V1.0, 1
S      Marcha_P:V3.1, 1
Network 71 //  DIN: Limpiar solicitud P->E al finalizar
// Acuse de aviso para la solicitud atendida
// y envio de solicitud de marcha para la unidad de Ensamblaje
LD     T_Tarea_Fin:M6.7
A      Ctx_Tarea_PE:M7.1
R      P2_Req_P_E:M0.2, 1
S      Ack_PE:V3.0, 1
S      Marcha_E:V5.1, 1
Network 72 // DIN: Limpiar solicitud E->S al finalizar
//  Acuse de aviso para la solicitud atendida
// y envio de solicitud de marcha para la unidad de Seleccion
LD     T_Tarea_Fin:M6.7
A      Ctx_Tarea_ES:M7.2
R      P3_Req_E_S:M0.3, 1
S      Ack_ES:V5.0, 1
S      Marcha_S:V7.1, 1
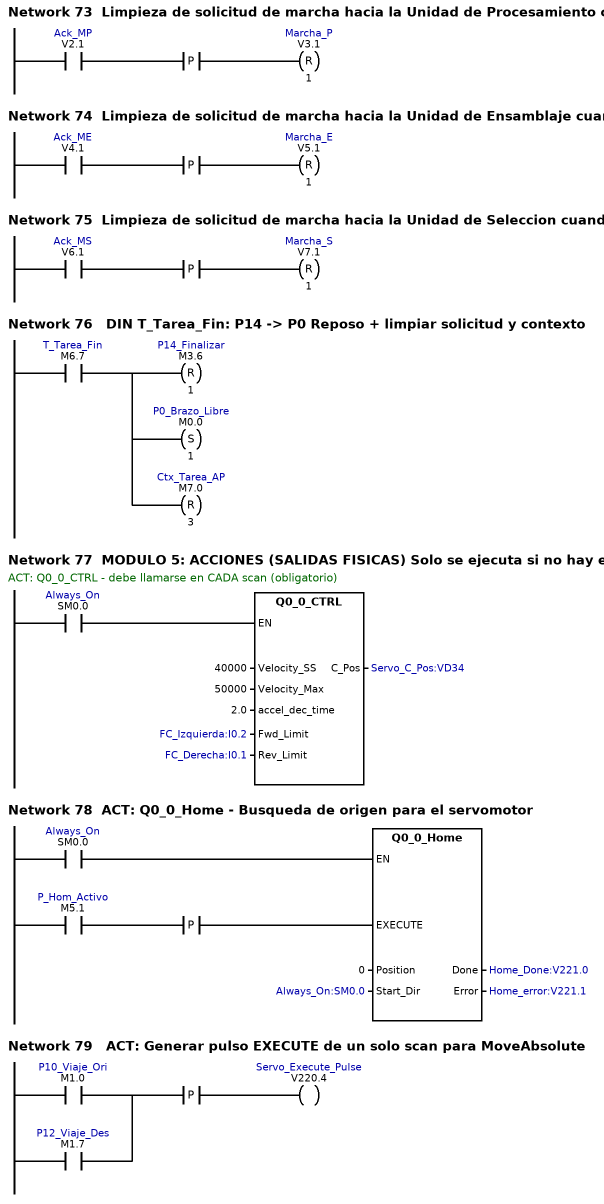
Network 73 // Limpieza de solicitud de marcha hacia la Unidad de Procesamiento cuando ha sido atendida
LD     Ack_MP:V2.1
EU
R      Marcha_P:V3.1, 1
Network 74 // Limpieza de solicitud de marcha hacia la Unidad de Ensamblaje cuando ha sido atendida
LD     Ack_ME:V4.1
EU
R      Marcha_E:V5.1, 1
Network 75 // Limpieza de solicitud de marcha hacia la Unidad de Seleccion cuando ha sido atendida
LD     Ack_MS:V6.1
EU
R      Marcha_S:V7.1, 1
Network 76 //  DIN T_Tarea_Fin: P14 -> P0 Reposo + limpiar solicitud y contexto
LD     T_Tarea_Fin:M6.7
R      P14_Finalizar:M3.6, 1
S      P0_Brazo_Libre:M0.0, 1
R      Ctx_Tarea_AP:M7.0, 3
Network 77 // MODULO 5: ACCIONES (SALIDAS FISICAS)
Solo se ejecuta si no hay emergencia (el JMP 2 lo omite).
Las llamadas a la libreria MAP_SERV van aqui.
// ACT: Q0_0_CTRL - debe llamarse en CADA scan (obligatorio)
LD     Always_On:SM0.0
CALL   Q0_0_CTRL:SBR3, 40000, 50000, 2.0, FC_Izquierda:I0.2, FC_Derecha:I0.1, Servo_C_Pos:VD34
Network 78 // ACT: Q0_0_Home - Busqueda de origen para el servomotor
LD     Always_On:SM0.0
=      L60.0
LD     P_Hom_Activo:M5.1
EU
=      L63.7
LD     L60.0
CALL   Q0_0_Home:SBR0, L63.7, 0, Always_On:SM0.0, Home_Done:V221.0, Home_error:V221.1
Network 79 //  ACT: Generar pulso EXECUTE de un solo scan para MoveAbsolute
LD     P10_Viaje_Ori:M1.0
O      P12_Viaje_Des:M1.7
EU
=      Servo_Execute_Pulse:V220.4
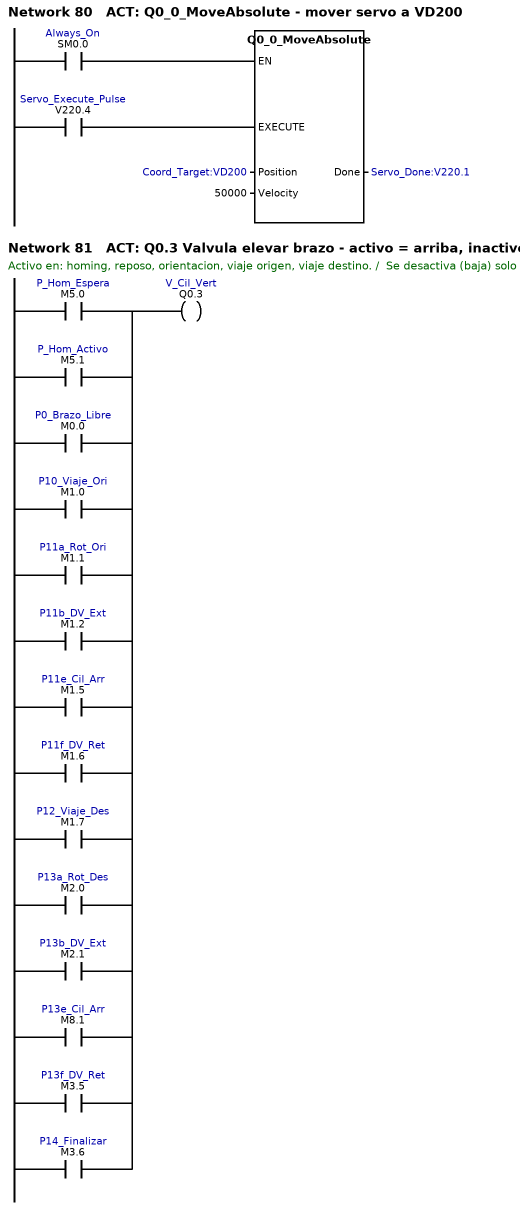
Network 80 //  ACT: Q0_0_MoveAbsolute - mover servo a VD200
LD     Always_On:SM0.0
=      L60.0
LD     Servo_Execute_Pulse:V220.4
=      L63.7
LD     L60.0
CALL   Q0_0_MoveAbsolute:SBR5, L63.7, Coord_Target:VD200, 50000, Servo_Done:V220.1
Network 81 //  ACT: Q0.3 Valvula elevar brazo - activo = arriba, inactivo = baja
//  Activo en: homing, reposo, orientacion, viaje origen, viaje destino.
//  Se desactiva (baja) solo en P11c y P13c (pasos de bajar).
// borrados: m2.4
LD     P_Hom_Espera:M5.0
O      P_Hom_Activo:M5.1
O      P0_Brazo_Libre:M0.0
O      P10_Viaje_Ori:M1.0
O      P11a_Rot_Ori:M1.1
O      P11b_DV_Ext:M1.2
O      P11e_Cil_Arr:M1.5
O      P11f_DV_Ret:M1.6
O      P12_Viaje_Des:M1.7
O      P13a_Rot_Des:M2.0
O      P13b_DV_Ext:M2.1
O      P13e_Cil_Arr:M8.1
O      P13f_DV_Ret:M3.5
O      P14_Finalizar:M3.6
=      V_Cil_Vert:Q0.3
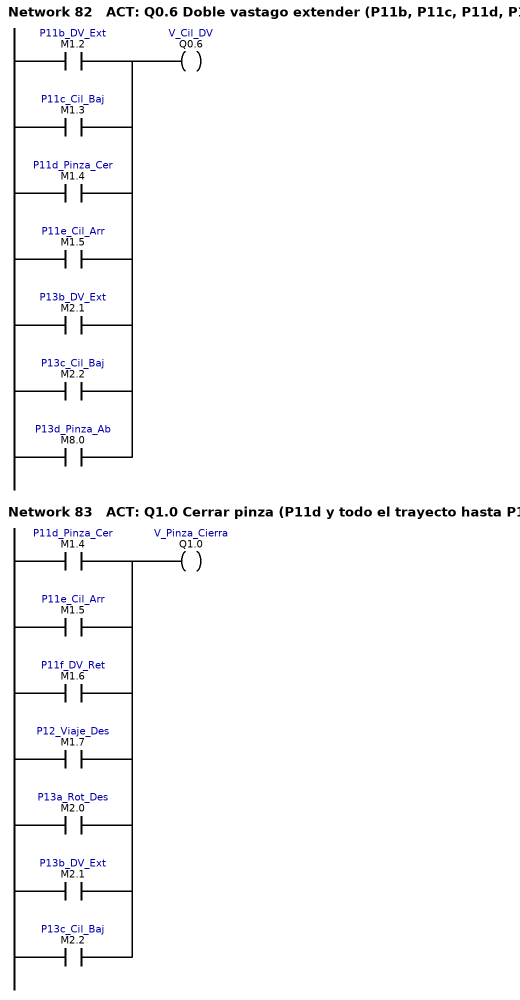
Network 82 //  ACT: Q0.6 Doble vastago extender (P11b, P11c, P11d, P13b, P13c, P13d)
LD     P11b_DV_Ext:M1.2
O      P11c_Cil_Baj:M1.3
O      P11d_Pinza_Cer:M1.4
O      P11e_Cil_Arr:M1.5
O      P13b_DV_Ext:M2.1
O      P13c_Cil_Baj:M2.2
O      P13d_Pinza_Ab:M8.0
=      V_Cil_DV:Q0.6
Network 83 //  ACT: Q1.0 Cerrar pinza (P11d y todo el trayecto hasta P13c)
LD     P11d_Pinza_Cer:M1.4
O      P11e_Cil_Arr:M1.5
O      P11f_DV_Ret:M1.6
O      P12_Viaje_Des:M1.7
O      P13a_Rot_Des:M2.0
O      P13b_DV_Ext:M2.1
O      P13c_Cil_Baj:M2.2
=      V_Pinza_Cierra:Q1.0
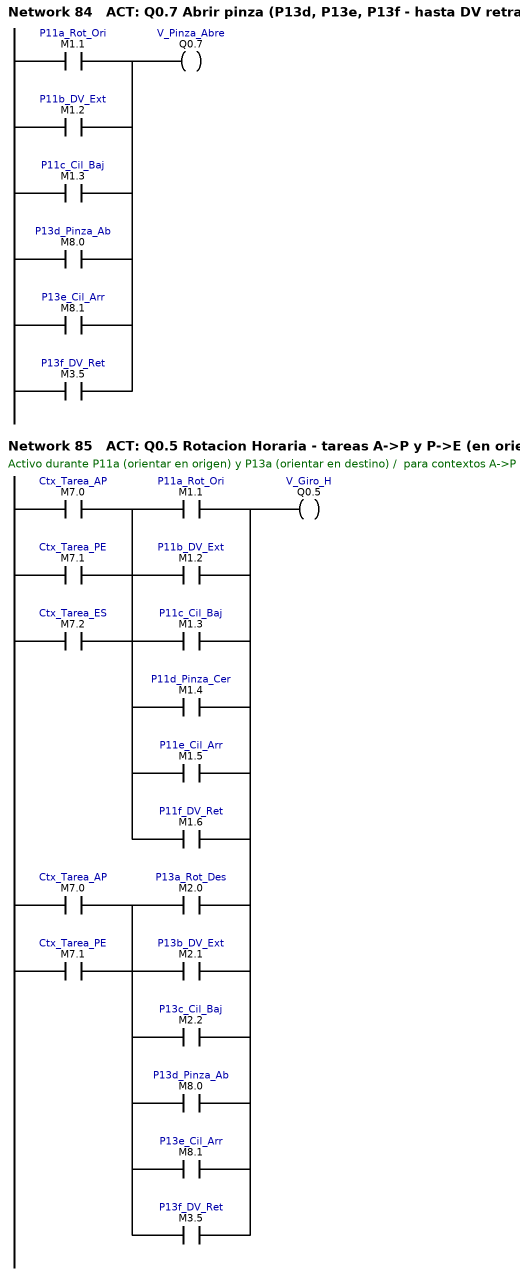
Network 84 //  ACT: Q0.7 Abrir pinza (P13d, P13e, P13f - hasta DV retraido)
LD     P11a_Rot_Ori:M1.1
O      P11b_DV_Ext:M1.2
O      P11c_Cil_Baj:M1.3
O      P13d_Pinza_Ab:M8.0
O      P13e_Cil_Arr:M8.1
O      P13f_DV_Ret:M3.5
=      V_Pinza_Abre:Q0.7
Network 85 //  ACT: Q0.5 Rotacion Horaria - tareas A->P y P->E (en orientacion de ambos extremos)
//  Activo durante P11a (orientar en origen) y P13a (orientar en destino)
//  para contextos A->P (M7.0) y P->E (M7.1).
//  Para E->S (M7.2): horario en origen, antihorario en destino.
LD     Ctx_Tarea_AP:M7.0
O      Ctx_Tarea_PE:M7.1
O      Ctx_Tarea_ES:M7.2
LD     P11a_Rot_Ori:M1.1
O      P11b_DV_Ext:M1.2
O      P11c_Cil_Baj:M1.3
O      P11d_Pinza_Cer:M1.4
O      P11e_Cil_Arr:M1.5
O      P11f_DV_Ret:M1.6
ALD
LD     Ctx_Tarea_AP:M7.0
O      Ctx_Tarea_PE:M7.1
LD     P13a_Rot_Des:M2.0
O      P13b_DV_Ext:M2.1
O      P13c_Cil_Baj:M2.2
O      P13d_Pinza_Ab:M8.0
O      P13e_Cil_Arr:M8.1
O      P13f_DV_Ret:M3.5
ALD
OLD
=      V_Giro_H:Q0.5
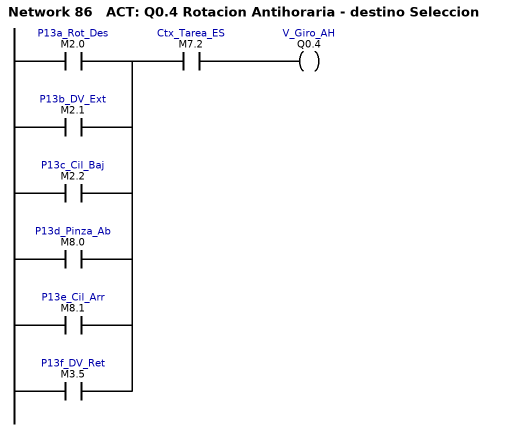
Network 86 //  ACT: Q0.4 Rotacion Antihoraria - destino Seleccion
// ===========================================================
// SENALIZACION
// ===========================================================
LD     P13a_Rot_Des:M2.0
O      P13b_DV_Ext:M2.1
O      P13c_Cil_Baj:M2.2
O      P13d_Pinza_Ab:M8.0
O      P13e_Cil_Arr:M8.1
O      P13f_DV_Ret:M3.5
A      Ctx_Tarea_ES:M7.2
=      V_Giro_AH:Q0.4
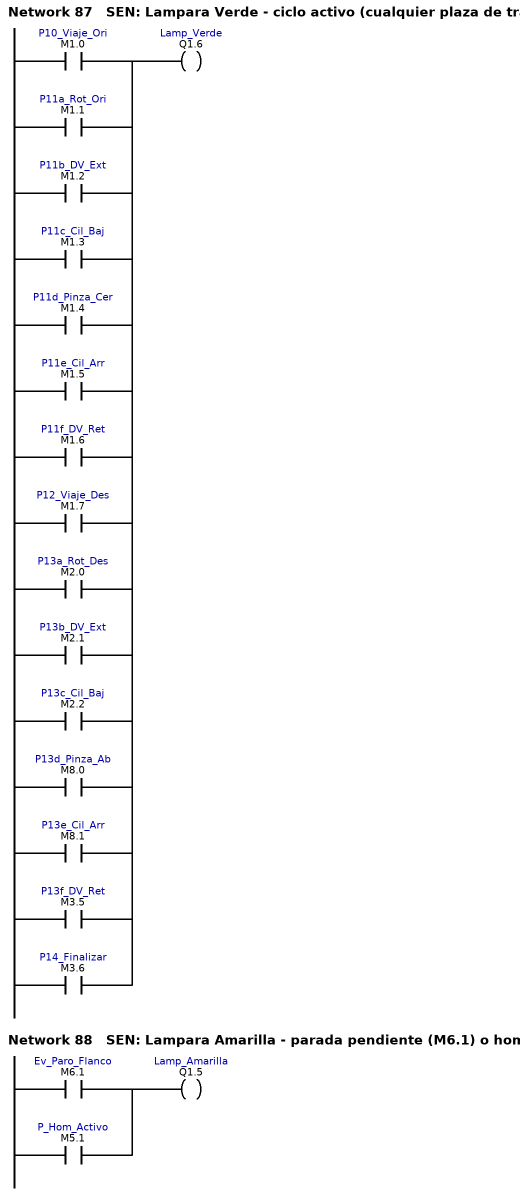
Network 87 //  SEN: Lampara Verde - ciclo activo (cualquier plaza de trabajo)
LD     P10_Viaje_Ori:M1.0
O      P11a_Rot_Ori:M1.1
O      P11b_DV_Ext:M1.2
O      P11c_Cil_Baj:M1.3
O      P11d_Pinza_Cer:M1.4
O      P11e_Cil_Arr:M1.5
O      P11f_DV_Ret:M1.6
O      P12_Viaje_Des:M1.7
O      P13a_Rot_Des:M2.0
O      P13b_DV_Ext:M2.1
O      P13c_Cil_Baj:M2.2
O      P13d_Pinza_Ab:M8.0
O      P13e_Cil_Arr:M8.1
O      P13f_DV_Ret:M3.5
O      P14_Finalizar:M3.6
=      Lamp_Verde:Q1.6
Network 88 //  SEN: Lampara Amarilla - parada pendiente (M6.1) o homing activo
LD     Ev_Paro_Flanco:M6.1
O      P_Hom_Activo:M5.1
=      Lamp_Amarilla:Q1.5
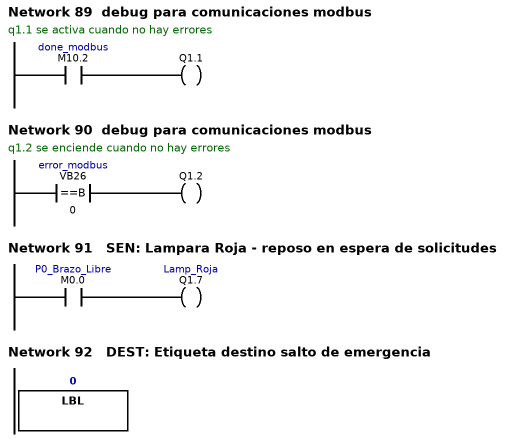
Network 89 // debug para comunicaciones modbus
// q1.1 se activa cuando no hay errores
LD     done_modbus:M10.2
=      Q1.1
Network 90 // debug para comunicaciones modbus
// q1.2 se enciende cuando no hay errores
LDB=   error_modbus:VB26, 0
=      Q1.2
Network 91 //  SEN: Lampara Roja - reposo en espera de solicitudes
LD     P0_Brazo_Libre:M0.0
=      Lamp_Roja:Q1.7
Network 92 //  DEST: Etiqueta destino salto de emergencia
LBL    0
END_ORGANIZATION_BLOCK

// SBR0: protected block, not included

// SBR1: protected block, not included

// SBR2: protected block, not included

// SBR3: protected block, not included

// SBR4: protected block, not included

// SBR5: protected block, not included

// SBR6: protected block, not included

// SBR7: protected block, not included

// SBR8: protected block, not included
